Yaskawa INFORM job: ROBOT.JBI

/JOB
//NAME ROBOT
///FOLDERNAME INNE
//POS
///NPOS 25,25,0,0,0,0
///TOOL 0
///POSTYPE PULSE
///PULSE
C00000=22847,-86279,-19911,-55793,83800,29326
C00001=-4565,-80787,-35612,-37946,82522,42300
C00002=-31769,-41742,-21367,-22143,102051,68513
C00003=-52548,-48866,-32950,-9514,97811,87456
C00004=-56817,-111136,-59948,-8579,47166,90656
C00005=-58920,-62811,-39707,4955,92932,68666
C00006=-77535,-81405,-48406,13178,80118,89934
C00007=23045,-72384,-20843,-42888,90113,67388
C00008=-48291,-132830,-47439,-308,10217,51311
C00009=-70665,-103353,-57481,15598,65309,41037
C00010=-61134,-104776,-48081,15795,57310,43408
C00011=7968,-83930,-33348,-27542,75221,74941
C00012=-66543,-123777,-43002,26020,31714,-1596
C00013=-89850,-75678,-31210,20714,84854,-38256
C00014=-76022,-54531,-20309,13758,96032,-49309
C00015=-33486,-99388,-47869,-2139,67701,-34730
C00016=-105730,-78237,-22372,32065,85248,-59983
C00017=-96413,-125141,-37954,44110,42530,-36872
C00018=12107,-50710,-12954,-20833,105862,3299
C00019=-42422,-56398,-23662,4009,101528,-18140
C00020=18052,-107220,-49365,1732,64372,-766
C00021=-70438,-62268,-3008,35164,96292,-60232
C00022=-115018,-117327,-27501,38193,69831,-52531
C00023=38403,-42328,-9494,-5182,104120,58380
C00024=130664,-84105,-14416,-40071,85398,83312
BC00000=246331,121646,575516
BC00001=246331,121646,575516
BC00002=246330,121646,575514
BC00003=246330,121646,575512
BC00004=246330,121646,575510
BC00005=246330,121645,575504
BC00006=246330,121645,575504
BC00007=246330,121645,575504
BC00008=246330,121645,575504
BC00009=246330,121645,575502
BC00010=246330,121645,575500
BC00011=246330,121645,575500
BC00012=246330,121645,575500
BC00013=246330,121645,575500
BC00014=246330,121645,575500
BC00015=246330,121645,575499
BC00016=246330,121645,575499
BC00017=246330,121645,575499
BC00018=246330,121645,575499
BC00019=246330,121645,575499
BC00020=246330,121644,575497
BC00021=246330,121644,575497
BC00022=246330,121644,575497
BC00023=246330,121644,575497
BC00024=246330,121644,575497
//INST
///DATE 2023/10/04 15:16
///ATTR SC,RW
///GROUP1 RB1,BS1
NOP
*1
MOVJ C00000 BC00000 VJ=0.78 PL=0
MOVJ C00001 BC00001 VJ=0.78 PL=0
MOVJ C00002 BC00002 VJ=0.78 PL=0
MOVJ C00003 BC00003 VJ=0.78 PL=0
MOVJ C00004 BC00004 VJ=0.78 PL=0
*2
MOVJ C00005 BC00005 VJ=0.78 PL=0
MOVJ C00006 BC00006 VJ=0.78 PL=0
MOVJ C00007 BC00007 VJ=0.78 PL=0
MOVJ C00008 BC00008 VJ=0.78 PL=0
MOVJ C00009 BC00009 VJ=0.78 PL=0
*3
MOVJ C00010 BC00010 VJ=0.78 PL=0
MOVJ C00011 BC00011 VJ=0.78 PL=0
MOVJ C00012 BC00012 VJ=0.78 PL=0
MOVJ C00013 BC00013 VJ=0.78 PL=0
MOVJ C00014 BC00014 VJ=0.78 PL=0
*4
MOVJ C00015 BC00015 VJ=0.78 PL=0
MOVJ C00016 BC00016 VJ=0.78 PL=0
MOVJ C00017 BC00017 VJ=0.78 PL=0
MOVJ C00018 BC00018 VJ=0.78 PL=0
MOVJ C00019 BC00019 VJ=0.78 PL=0
*5
MOVJ C00020 BC00020 VJ=0.78 PL=0
MOVJ C00021 BC00021 VJ=0.78 PL=0
MOVJ C00022 BC00022 VJ=0.78 PL=0
MOVJ C00023 BC00023 VJ=0.78 PL=0
MOVJ C00024 BC00024 VJ=0.78 PL=0
END
